PROGRAM PWM_valvulas
VAR
	
pwm1 : FB_CTRL_PWM_OUT;
pwm2 : FB_CTRL_PWM_OUT;
stParams                : ST_CTRL_PWM_OUT_PARAMS;

END_VAR

//parametrización PWM
stParams.bInstantPWMUpdate:=FALSE;
stParams.tPWMPeriod:=T#10MS;
stParams.tTaskCycleTime:=T#1MS;
pwm1(stParams:=stParams);
pwm1.eMode:=E_CTRL_MODE.eCTRL_MODE_ACTIVE;
pwm2(stParams:=stParams);
pwm2.eMode:=E_CTRL_MODE.eCTRL_MODE_ACTIVE;

//Cilindro 1
IF GVL.Cilindro1.regimen > 0 THEN
	pwm1.fPwmInput:=GVL.Cilindro1.regimen;
	IO.valv_alfa_mas:= pwm1.bPwmOutBitPos;
	IO.valv_alfa_menos:=0;
	GVL.Cilindro1.extendiendo:=TRUE;
	GVL.Cilindro1.retrayendo:=FALSE;
	GVL.Cilindro1.parado:=FALSE;
	ELSE IF GVL.Cilindro1.regimen < 0 THEN
			pwm1.fPwmInput:=-GVL.Cilindro1.regimen; //para mantenerlo positivo
			IO.valv_alfa_mas:= 0;
			IO.valv_alfa_menos:= pwm1.bPwmOutBitPos;
			GVL.Cilindro1.extendiendo:=FALSE;
			GVL.Cilindro1.retrayendo:=TRUE;
			GVL.Cilindro1.parado:=FALSE;
	ELSE 
	IO.valv_alfa_mas:= 0;
	IO.valv_alfa_menos:=0;
	GVL.Cilindro1.extendiendo:=FALSE;
	GVL.Cilindro1.retrayendo:=FALSE;
	GVL.Cilindro1.parado:=TRUE;
	END_IF 
END_IF

//Cilindro 2
IF GVL.Cilindro2.regimen > 0 THEN
	pwm2.fPwmInput:=GVL.Cilindro2.regimen;
	IO.valv_beta_mas:= pwm2.bPwmOutBitPos;
	IO.valv_beta_menos:= 0;
	GVL.Cilindro2.extendiendo:=TRUE;
	GVL.Cilindro2.retrayendo:=FALSE;
	GVL.Cilindro2.parado:=FALSE;
	ELSE IF GVL.Cilindro2.regimen < 0 THEN
			pwm2.fPwmInput:=-GVL.Cilindro2.regimen; //para mantenerlo positivo
			IO.valv_beta_mas:=0;
			IO.valv_beta_menos:= pwm2.bPwmOutBitPos;
			GVL.Cilindro2.extendiendo:=FALSE;
			GVL.Cilindro2.retrayendo:=TRUE;
			GVL.Cilindro2.parado:=FALSE;
	ELSE 
	IO.valv_beta_mas:=0;
	IO.valv_beta_menos:=0;
	GVL.Cilindro2.extendiendo:=FALSE;
	GVL.Cilindro2.retrayendo:=FALSE;
	GVL.Cilindro2.parado:=TRUE;
	END_IF 
END_IF

END_PROGRAM

(* stored: Version 1.1.0.1, ProductVersion 3.1.4024.4
   POU PWM_valvulas: Id {dd73676d-6682-49ad-bf70-d2556d73c910}, SpecialFunc None *)
